{attribute 'GeneratedUsingTerminal: EP2339-0021-0017'}
{attribute addProperty BoxType "EP2339-0021-0017"}
{attribute addProperty Description "EP2339-0021 16 Ch. Dig. Input/Output 24V, 0,5A, M8"}
{attribute addProperty Physics "YY"}
{attribute addProperty Id "Channel_1AT %I*Channel_830843C11Channel_2AT %I*Channel_830843C11Channel_3AT %I*Channel_830843C11Channel_4AT %I*Channel_830843C11Channel_5AT %I*Channel_830843C11Channel_6AT %I*Channel_830843C11Channel_7AT %I*Channel_830843C11Channel_8AT %I*Channel_830843C11Channel_9AT %I*Channel_830843C11Channel_10AT %I*Channel_830843C11Channel_11AT %I*Channel_830843C11Channel_12AT %I*Channel_830843C11Channel_13AT %I*Channel_830843C11Channel_14AT %I*Channel_830843C11Channel_15AT %I*Channel_830843C11Channel_16AT %I*Channel_830843C11Channel_17AT %Q*Channel_42CA91F71Channel_18AT %Q*Channel_42CA91F71Channel_19AT %Q*Channel_42CA91F71Channel_20AT %Q*Channel_42CA91F71Channel_21AT %Q*Channel_42CA91F71Channel_22AT %Q*Channel_42CA91F71Channel_23AT %Q*Channel_42CA91F71Channel_24AT %Q*Channel_42CA91F71Channel_25AT %Q*Channel_42CA91F71Channel_26AT %Q*Channel_42CA91F71Channel_27AT %Q*Channel_42CA91F71Channel_28AT %Q*Channel_42CA91F71Channel_29AT %Q*Channel_42CA91F71Channel_30AT %Q*Channel_42CA91F71Channel_31AT %Q*Channel_42CA91F71Channel_32AT %Q*Channel_42CA91F71WcStateAT %I*WcState_9091E0EB2InfoDataAT %I*InfoData_0A66F0098"}
{attribute addProperty CRC "3639210650"}
{attribute addProperty Size "42"}
TYPE EP2339_D8E9F29A EXTENDS EtcSlaveBoxBase_77A0E4A7 :
STRUCT
	{attribute addProperty Name "Channel_1"}
	Channel_1 : Channel_830843C1;
	{attribute addProperty Name "Channel_2"}
	Channel_2 : Channel_830843C1;
	{attribute addProperty Name "Channel_3"}
	Channel_3 : Channel_830843C1;
	{attribute addProperty Name "Channel_4"}
	Channel_4 : Channel_830843C1;
	{attribute addProperty Name "Channel_5"}
	Channel_5 : Channel_830843C1;
	{attribute addProperty Name "Channel_6"}
	Channel_6 : Channel_830843C1;
	{attribute addProperty Name "Channel_7"}
	Channel_7 : Channel_830843C1;
	{attribute addProperty Name "Channel_8"}
	Channel_8 : Channel_830843C1;
	{attribute addProperty Name "Channel_9"}
	Channel_9 : Channel_830843C1;
	{attribute addProperty Name "Channel_10"}
	Channel_10 : Channel_830843C1;
	{attribute addProperty Name "Channel_11"}
	Channel_11 : Channel_830843C1;
	{attribute addProperty Name "Channel_12"}
	Channel_12 : Channel_830843C1;
	{attribute addProperty Name "Channel_13"}
	Channel_13 : Channel_830843C1;
	{attribute addProperty Name "Channel_14"}
	Channel_14 : Channel_830843C1;
	{attribute addProperty Name "Channel_15"}
	Channel_15 : Channel_830843C1;
	{attribute addProperty Name "Channel_16"}
	Channel_16 : Channel_830843C1;
	{attribute addProperty Name "Channel_17"}
	Channel_17 : Channel_42CA91F7;
	{attribute addProperty Name "Channel_18"}
	Channel_18 : Channel_42CA91F7;
	{attribute addProperty Name "Channel_19"}
	Channel_19 : Channel_42CA91F7;
	{attribute addProperty Name "Channel_20"}
	Channel_20 : Channel_42CA91F7;
	{attribute addProperty Name "Channel_21"}
	Channel_21 : Channel_42CA91F7;
	{attribute addProperty Name "Channel_22"}
	Channel_22 : Channel_42CA91F7;
	{attribute addProperty Name "Channel_23"}
	Channel_23 : Channel_42CA91F7;
	{attribute addProperty Name "Channel_24"}
	Channel_24 : Channel_42CA91F7;
	{attribute addProperty Name "Channel_25"}
	Channel_25 : Channel_42CA91F7;
	{attribute addProperty Name "Channel_26"}
	Channel_26 : Channel_42CA91F7;
	{attribute addProperty Name "Channel_27"}
	Channel_27 : Channel_42CA91F7;
	{attribute addProperty Name "Channel_28"}
	Channel_28 : Channel_42CA91F7;
	{attribute addProperty Name "Channel_29"}
	Channel_29 : Channel_42CA91F7;
	{attribute addProperty Name "Channel_30"}
	Channel_30 : Channel_42CA91F7;
	{attribute addProperty Name "Channel_31"}
	Channel_31 : Channel_42CA91F7;
	{attribute addProperty Name "Channel_32"}
	Channel_32 : Channel_42CA91F7;
	{attribute addProperty Name "WcState"}
	WcState : WcState_9091E0EB;
	{attribute addProperty Name "InfoData"}
	InfoData : InfoData_0A66F009;
END_STRUCT
END_TYPE

(* stored: Version 1.2.0.0, ProductVersion 3.1.4024.9
   DUT EP2339_D8E9F29A: Id {05e0c0a3-9ed7-4a54-bde7-c14dc4808e54} *)
